{attribute 'qualified_only'}
{attribute 'strict'}
TYPE EFeedbackMsgPolarisationELL14K :
(
	PositionMsg := 10,
    IdMsg,
	CalibMsg,
    CustomMsg
);
END_TYPE

(* stored: Version 1.1.0.1, ProductVersion 3.1.4024.10
   DUT EFeedbackMsgPolarisationELL14K: Id {eac2379b-7585-4975-b323-4e8f9d44ead2} *)
